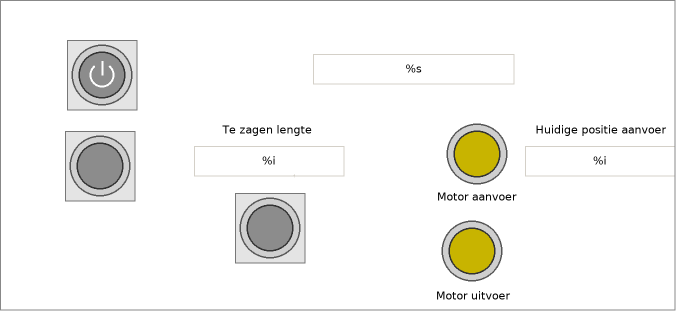
VISUALIZATION Visualization  // 676x311
    PushSwitch (65,131 70x70), variable: MAIN.Initialiseren, behaviour: TOGGLE, style: Switch-PushSwitch-Gray
    Textfield (313,54 201x30), "%s", text variable: MAIN.Status
    Lamp1 (442,119 70x70), variable: GVL.MotorInvoer, style: Lamp-Lamp1-Yellow
    Lamp1 (437,216 70x70), variable: GVL.MotorUitvoer, style: Lamp-Lamp1-Yellow
    Label (402,182 150x30), "Motor aanvoer"
    Label (398,281 150x30), "Motor uitvoer"
    Textfield (194,146 150x30), "%i", text variable: GVL.ZaagLengte, invisible if: NOT (MAIN.Initialisatie_voltooid)
        OnMouseClick: write GVL.ZaagLengte via VisuDialogs.Numpad, min 1, max 6000
    Label (194,115 150x30), "Te zagen lengte", invisible if: NOT (MAIN.Initialisatie_voltooid)
    Textfield (525,146 150x30), "%i", text variable: GVL.HuidigePositieAanvoer
    Label (526,115 150x30), "Huidige positie aanvoer"
    PowerSwitch (67,40 70x70), variable: MAIN.Power, behaviour: TOGGLE, style: Switch-PowerSwitch-Gray
    Textfield (294,174 0x3)
    PushSwitch (235,193 70x70), variable: GVL.StartAanvoer, behaviour: TOGGLE, style: Switch-PushSwitch-Gray
END_VISUALIZATION

(* stored: Version 1.1.0.1, ProductVersion 3.1.4024.12
   Visu Visualization: Id {fbc54d82-2f12-437e-af0a-8ed45a203fbc} *)
